KUKA KRL program: chk_w11_grp1_clo.src

&ACCESS RVO3
&COMMENT Axor 913 Z1.1_Z1.2
DEF chk_w11_grp1_clo( )
; Check gripper AXOR 913 CLOSE Z1.1/2
;//---- Start User-------

$TIMER[10] = 0
$TIMER_STOP[10] = FALSE

WAIT FOR ($IN[526] AND $IN[528])
WAIT FOR (NOT $IN[525] AND NOT $IN[527])

$TIMER_STOP[10] = TRUE
$TIMER[10] = 0

;//---- End User---------
END
